ABB RAPID module: main.mod

MODULE MainModule
GLOBAL VAR intnum test_int
LOCAL VAR robtarget p1 = p:{{444.592163546,-0.012366435,562.885466728},{0.642890516,0.000011540,0.765958083,-0.000008196}}{cfg -1,0,-1,0}{EJ 0.000000000,0.000000000,0.000000000,0.000000000,0.000000000,0.000000000}
LOCAL VAR robtarget p2 = p:{{406.322726251,334.967342629,32.137701315},{-0.018301280,-0.327458252,0.944444310,-0.021473281}}{cfg 0,-1,0,0}{EJ 0.000000000,0.000000000,0.000000000,0.000000000,0.000000000,0.000000000}
LOCAL VAR robtarget p3 = p:{{406.327318602,334.970726404,398.112972108},{-0.018332796,-0.327460720,0.944442425,-0.021491655}}{cfg 0,-1,0,0}{EJ 0.000000000,0.000000000,0.000000000,0.000000000,0.000000000,0.000000000}
LOCAL VAR robtarget p4 = p:{{406.996750170,-344.976978114,390.531910622},{-0.025825354,-0.327485510,0.944191478,-0.024264042}}{cfg -1,-1,-1,0}{EJ 0.000000000,0.000000000,0.000000000,0.000000000,0.000000000,0.000000000}
LOCAL VAR robtarget p5 = p:{{406.986658982,-344.958435970,85.026482811},{-0.025828364,-0.327501842,0.944186337,-0.024240465}}{cfg -1,-1,-1,0}{EJ 0.000000000,0.000000000,0.000000000,0.000000000,0.000000000,0.000000000}
LOCAL VAR robtarget p6 = p:{{406.983103706,-344.951417839,272.002632681},{-0.025848482,-0.327498467,0.944187605,-0.024215228}}{cfg -1,-1,-1,0}{EJ 0.000000000,0.000000000,0.000000000,0.000000000,0.000000000,0.000000000}
LOCAL VAR robtarget p7 = p:{{398.014291991,-0.002355527,629.485470635},{0.707088996,-0.000013333,0.707124566,-0.000017517}}{cfg -1,-1,-1,0}{EJ 0.000000000,0.000000000,0.000000000,0.000000000,0.000000000,0.000000000}

GLOBAL PROC main()
	WHILE(TRUE)
		Wait 0.01
		CONNECT test_int WITH test
		ISignalDI \Single,RobotDI1,0,test_int
	ENDWHILE
ENDPROC

GLOBAL TRAP test
	StopMove
	StorePath
    p7=CRobT()
	MoveJ p1,v100,fine,tool0
	MoveJ p2,v200,fine,tool0
	Wait 2
	MoveL p3,v200,z50,tool0
	MoveL p4,v200,z50,tool0
	MoveL p5,v200,fine,tool0
	Wait 2
	MoveL p6,v200,fine,tool0
	MoveJ p7,v200,fine,tool0
	RobotDO1==TRUE
	RestoPath
	StartMove
ENDTRAP
ENDMODULE
